Fanuc KAREL source: SEND_EVENTPC.kl

PROGRAM T
%NOLOCKGROUP
VAR
 v0 : INTEGER
 v1 : INTEGER
BEGIN
 SEND_EVENTPC(v0, v1)
END T
